INTERFACE IInspector

PROPERTY Busy : BOOL
GET
END_GET
END_PROPERTY

PROPERTY Done : BOOL
GET
END_GET
END_PROPERTY

METHOD OnFail : IOnFail
END_METHOD

PROPERTY OverInspected : BOOL
GET
END_GET
END_PROPERTY

PROPERTY Result : eInspectorResult
GET
END_GET
END_PROPERTY

METHOD UpdateComprehensiveResult : IInspector
VAR_IN_OUT
    inoResult : TcoComprehensiveResult;
END_VAR
END_METHOD

END_INTERFACE

(* stored: Version 1.1.0.1, ProductVersion 3.1.4024.9
   Itf IInspector: Id {0cbe9e39-d5a4-05af-17ce-7965efd20de3}
   Property Busy: Id {b32bf15d-c374-0d51-2e79-45bad14701d4}
   Get Get: Id {ebd05d89-2b98-0f79-0951-70a8ea77ee5c}
   Property Done: Id {619d20fa-40bc-0c73-013c-9ce9a7b16b05}
   Get Get: Id {dda1cead-ae16-0ba2-2984-226a50200b84}
   Method OnFail: Id {ac3abd9c-363c-070f-178a-504f9b7741ff}
   Property OverInspected: Id {8def8039-9580-0717-1f67-557c2ea921c0}
   Get Get: Id {7ec14b78-0f82-0a30-2aad-7349dddb37bc}
   Property Result: Id {059b95a9-368b-016b-1e77-bc829a9a2a15}
   Get Get: Id {11bcb09e-df05-0600-3fcc-c1e8eab49bfc}
   Method UpdateComprehensiveResult: Id {5d6cf906-2212-0e3f-182f-3c47b27fe0e1} *)
